FUNCTION_BLOCK SwitchToMaintenance
VAR_INPUT
END_VAR
VAR_OUTPUT
END_VAR
VAR
	SwitchToMaintenance : BOOL;
END_VAR

IF SwitchToMaintenance THEN 
	GoToBasicPosition();
END_IF

METHOD PUBLIC GoToBasicPosition : BOOL
VAR_INPUT
END_VAR
GoToBasicPosition := 0;
END_METHOD

END_FUNCTION_BLOCK

(* stored: Version 1.1.0.1, ProductVersion 3.1.4020.12
   POU SwitchToMaintenance: Id {60d55301-fa8c-4a1a-8833-0db841841e56}, SpecialFunc None
   Method GoToBasicPosition: Id {716b087d-1bc5-440d-a3f4-f48b1f107be7} *)
